Fanuc KAREL source: kt00336.KL

-- PROVISIONAL review KL for V1013-1; original PC SHA256 165b99eb11a4b85a7f498307c7af127f50c182e5eb3783f22ad2ae9d74c2ab39
-- Incomplete behavior may be omitted. Consult companion uncertainty JSON. Do not deploy.
PROGRAM KT00336
%NOLOCKGROUP
VAR
  R1 : REAL
  OUT : BOOLEAN
-- UNRESOLVED_DECL H2 type=002017
BEGIN
  -- UNRESOLVED_PC offsets 5-16; opcodes 2E,23
  -- UNRESOLVED_PC offsets 21-35; opcodes 2E,22,9D,33,B4
  -- UNRESOLVED_PC offsets 40-63; opcodes 21,22,9D,33,B3,64,6F,23
  -- UNRESOLVED_PC offsets 68-72; opcodes 7F
END KT00336
